FUNCTION_BLOCK FB_PCMChiller EXTENDS FB_ActuatorContinous
VAR_INPUT
	fExternalTemperature : REAL; 
	nControlModeAutomatic : E_PCMControlMode;
END_VAR
VAR_OUTPUT
END_VAR
VAR
	
	{attribute 'OPC.UA.DA' := '1'}
	localState : ST_pcmChillerState;
	//default parameters
	localDefaultParameters : ST_pcmChillerDefaultParameters;
	//I/O Links
	nRemoteControl_OUT AT %Q* : DINT;
	nSetPointMediumTemperature_OUT AT %Q* : LREAL;
	fAmbientTemperature_IN AT %I* : LREAL;
	fMediumOutletTemperature_IN AT %I* : LREAL; 
	fCoolingCapacity_IN AT %I* : DINT; 
	fCoolingEER_IN AT %I* : LREAL; 
	fFlowValue_IN AT %I* : LREAL; 
	fFanValue_IN AT %I* : DINT; 
	fCompressorSpeed_IN AT %I* : DINT; 
	fEEVValue_IN AT %I* : LREAL; 
	fEEVPosition_IN AT %I* : DINT; 
	fInputPower_IN AT %I* : DINT; 
	fEnvironmentTemperature_IN AT %I* : LREAL;
	
	//internal variables
	nControlMode : E_PCMControlMode;
END_VAR

MAIN();

METHOD GetState : BOOL
VAR_INPUT
END_VAR
//control state


//setpoint state
setPointState.fOperatingPoint := fExternalTemperature; //adjust fExternalTemperature to the right variable
setPointState.sOperatingPointUnit := 'degreeC'; 
fOperatingPoint := fExternalTemperature; 

//local state
localState.fAmbientTemperature := fAmbientTemperature_IN;
localState.fCompressorSpeed := fCompressorSpeed_IN;
localState.fCoolingCapacity := fCoolingCapacity_IN; 
localState.fCoolingEER := fCoolingEER_IN; 
localState.fEEVPosition := fEEVPosition_IN; 
localState.fEEVValue := fEEVValue_IN; 
localState.fEnvironmentTemperature := fEnvironmentTemperature_IN; 
localState.fFanValue := fFanValue_IN; 
localState.fFlowValue := fFlowValue_IN; 
localState.fInputPower := fInputPower_IN;
localState.fMediumOutletTemperature := fMediumOutletTemperature_IN;
END_METHOD

METHOD PROTECTED  SetSetPointLimits : BOOL
VAR_INPUT
END_VAR
aSetPointLimits[1] := localDefaultParameters.aSetPointLimitsTemperature[1];
aSetPointLimits[2] := localDefaultParameters.aSetPointLimitsTemperature[2];
END_METHOD

METHOD SetState : BOOL
VAR_INPUT
END_VAR
setPointState.fSetPoint := fSetPoint;
setPointState.aSetPointLimits := aSetPointLimits;
setPointState.sSetPointUnit := 'degreeC';


nSetPointMediumTemperature_OUT := fSetPoint;

IF bSetStatusOn THEN
	CASE nControlMode OF
		0: //cooling mode
		nRemoteControl_OUT := 0;
		
		1: //pump mode
		nRemoteControl_OUT := 2;
	END_CASE
ELSE
	nRemoteControl_OUT := 1; //Stand-By
END_IF;
END_METHOD

PROPERTY ST_DefaultParameters : REFERENCE TO ST_pcmChillerDefaultParameters
GET
ST_DefaultParameters REF= localDefaultParameters;
END_GET
SET
localDefaultParameters := ST_DefaultParameters;
END_SET
END_PROPERTY

END_FUNCTION_BLOCK

(* stored: Version 1.1.0.1, ProductVersion 3.1.4024.10
   POU FB_PCMChiller: Id {6d6159d2-75d3-4fc2-803c-5a2854a50767}, SpecialFunc None
   Method GetState: Id {d66ab647-cb72-495a-adc6-69e68b5651cf}
   Method SetSetPointLimits: Id {bfb24d2f-5849-48b8-bbf8-f6f04ee35cf3}
   Method SetState: Id {ec1b9726-e7f0-4f1e-85e0-77391a5577b6}
   Property ST_DefaultParameters: Id {89822b66-c4d4-4758-8808-1dc9a87e88d5}
   Get Get: Id {1462475c-944f-4d4a-9089-ef70c837b5b6}
   Set Set: Id {281901a6-caa9-4b5a-bd1e-70ddd648e277} *)
